(* CODESYS project 2.project

Project tree, tasks and I/O mapping:
  Device : CODESYS Control Win V3, 3S - Smart Software Solutions GmbH, order no. 305021, version 3.5.11.30
    application Application
      libraries: Standard, * (System)
      task MainTask (cyclic, interval t#20ms, priority 1) calls PLC_PRG
      program PLC_PRG [LD]
*)

// Device/Application/PLC_PRG
PROGRAM PLC_PRG
VAR
	BT1: BOOL;
	L1: BOOL;
	BT2: BOOL;
	L2: BOOL;
	BT3: BOOL;
	L3: BOOL;
	AUX: BOOL;
END_VAR

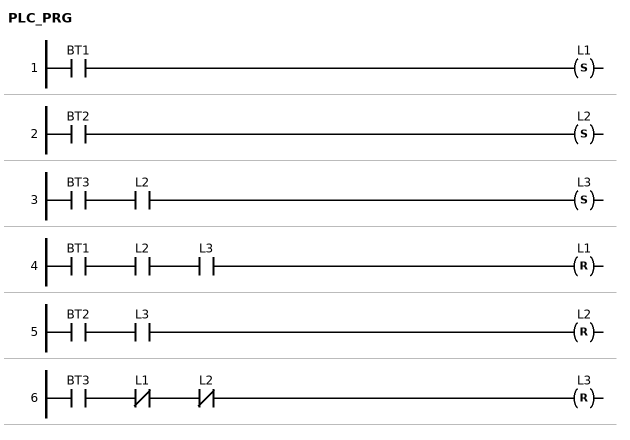
// NETWORK 1
L1 S= BT1;

// NETWORK 2
L2 S= BT2;

// NETWORK 3
L3 S= BT3 AND L2;

// NETWORK 4
L1 R= BT1 AND L2 AND L3;

// NETWORK 5
L2 R= BT2 AND L3;

// NETWORK 6
L3 R= BT3 AND NOT L1 AND NOT L2;

END_PROGRAM
